Yaskawa INFORM job: KRIS3(-160_-90)54.JBI

/JOB
//NAME KRIS3(-160_-90)54
//POS
///NPOS 266,266,266,20,0,0
///TOOL 0
///POSTYPE PULSE
///PULSE
C00000=-36470,-76528,-106815,19279,71473,77234
C00001=-136908,-99459,-124829,20670,71348,76391
C00002=-134470,-76528,-106815,19279,71473,77234
C00003=-159578,-94739,-111578,14965,102577,71346
C00004=-157566,-87256,-71357,3912,80960,68626
C00005=-176880,-68125,-57902,5422,83635,62119
C00006=-177907,-68461,-55745,5507,82211,61705
C00007=-177907,-68063,-54493,5513,81648,61681
C00008=-177907,-68139,-54730,5512,81754,61686
C00009=-178677,-69433,-55362,5571,81531,61412
C00010=-178017,-68613,-55721,5516,82126,61665
C00011=-169648,-85474,-89038,4887,93378,64966
C00012=-163611,-44630,-68122,4506,101126,67267
C00013=-165231,-48362,-64740,4579,97228,66587
C00014=-165334,-48746,-64513,4584,96897,66540
C00015=-165334,-48893,-63576,4578,96247,66515
C00016=-165334,-48863,-63784,4579,96390,66520
C00017=-165646,-49802,-64330,4606,96263,66409
C00018=-165334,-48746,-64513,4584,96897,66540
C00019=-140979,-108094,-110643,2385,93763,74547
C00020=-140979,-108094,-110643,2385,93763,74547
C00021=-140979,-108094,-110643,2385,93763,74547
C00022=-140979,-108094,-110643,2385,93763,74547
C00023=-140979,-108246,-109289,2383,92853,74530
C00024=-140979,-108231,-109453,2383,92961,74533
C00025=-141280,-110659,-110301,2409,92244,74420
C00026=-140979,-108094,-110643,2385,93763,74547
C00027=-156700,-55897,-85418,-8720,99373,67438
C00028=-156898,-58036,-83987,-8629,97394,67513
C00029=-156898,-58722,-82817,-8603,96332,67586
C00030=-156898,-58622,-82997,-8608,96491,67574
C00031=-157341,-60416,-83948,-8523,96115,67457
C00032=-156898,-58036,-83987,-8629,97394,67513
C00033=-161369,-86849,-99090,4273,98390,67906
C00034=-167909,-84037,-82934,-3708,84523,64877
C00035=-168571,-85124,-82512,-3609,83677,64677
C00036=-168571,-84898,-80901,-3613,82804,64704
C00037=-168571,-84936,-81149,-3613,82937,64700
C00038=-169203,-86467,-81802,-3516,82525,64499
C00039=-168571,-85124,-82512,-3609,83677,64677
C00040=-165600,-121955,-98284,-4061,74695,65975
C00041=-174461,-109455,-70225,-9835,59183,64105
C00042=-175080,-109402,-69148,-9749,58483,63930
C00043=-175080,-108469,-67668,-9792,58058,63969
C00044=-175080,-108628,-67921,-9785,58130,63962
C00045=-176152,-109889,-68298,-9565,57596,63593
C00046=-175080,-109402,-69148,-9749,58483,63930
C00047=-145436,-132582,-96247,-390,75065,72870
C00048=-145436,-132678,-96385,-390,75101,72870
C00049=-145436,-153478,-122593,-390,33069,72870
C00050=-145436,-153478,-122593,-390,33069,72870
C00051=-145875,-137224,-99164,-151,44123,76557
C00052=-145875,-137224,-99164,3186,26783,75636
C00053=-145875,-137224,-99164,3186,26783,75636
C00054=-126920,-141995,-100488,-14842,27437,88451
C00055=-126921,-139435,-97257,-15195,26791,88624
C00056=-126921,-140260,-98306,-15082,27005,88567
C00057=-126657,-136107,-97292,-14665,28515,88375
C00058=-126920,-141995,-100488,-14842,27437,88451
C00059=-153689,-122615,-92358,-7246,28662,82796
C00060=-153689,-122359,-91923,-7277,28527,82812
C00061=-153689,-121251,-90046,-7417,27945,82882
C00062=-153689,-121596,-90629,-7373,28125,82859
C00063=-152562,-118169,-89603,-8504,29355,83484
C00064=-153689,-122359,-91923,-7277,28527,82812
C00065=-153734,-144670,-102026,12528,26386,79802
C00066=-148920,-141423,-91163,14854,15551,80235
C00067=-148967,-137496,-86916,15534,14983,79917
C00068=-147891,-134819,-86332,12174,15793,81580
C00069=-148428,-136185,-86633,13817,15374,80764
C00070=-148428,-134667,-84751,14154,15007,80609
C00071=-149705,-139389,-87494,17948,14535,78726
C00072=-140769,-160579,-91179,72763,19950,46602
C00073=-129302,-154781,-89703,59410,13959,54584
C00074=-128993,-152913,-89439,56337,14227,56040
C00075=-129214,-154274,-89633,58559,14027,54988
C00076=-129214,-151990,-87339,59384,13900,54610
C00077=-129539,-156129,-91089,59119,14177,54682
C00078=-130002,-156587,-91482,58522,14566,54861
C00079=-131612,-152018,-92345,56188,18115,55777
C00080=-137260,-138866,-133764,10166,31487,76482
C00081=-31464,-162597,-133764,10166,12061,76482
C00082=11401,-148032,-125425,11667,35640,75771
C00083=126225,-114648,-117375,36487,17100,65054
C00084=160935,-140983,-109640,13468,75088,74332
C00085=169853,-118963,-84593,12681,69660,-86771
C00086=166041,-110678,-74459,13320,68331,-88303
C00087=166223,-108797,-70951,13405,67140,-88373
C00088=166223,-107663,-69097,13458,66595,-88438
C00089=166223,-107867,-69431,13449,66693,-88427
C00090=167322,-109580,-69957,13369,65975,-88109
C00091=166243,-109210,-71582,13386,67309,-88347
C00092=169217,-106350,-70409,12947,67561,-87233
C00093=169217,-106256,-70250,12951,67512,-87238
C00094=169217,-105112,-68312,13006,66921,-87306
C00095=169217,-105283,-68599,12998,67008,-87297
C00096=170397,-106999,-69102,12897,66265,-86949
C00097=167930,-107758,-71144,13135,67501,-87709
C00098=168330,-125239,-100831,12460,76505,-86600
C00099=155830,-85289,-85709,13656,89459,-89593
C00100=155617,-85922,-82565,13677,87294,-89905
C00101=155617,-85683,-81004,13681,86480,-89993
C00102=155617,-85728,-81276,13680,86620,-89979
C00103=156391,-88450,-82422,13606,85816,-89798
C00104=155763,-86416,-82528,13661,87001,-89886
C00105=155923,-87175,-84120,13644,87549,-89771
C00106=155609,-85916,-82709,13676,87386,-89897
C00107=155609,-85729,-81437,13679,86718,-89971
C00108=155609,-85763,-81652,13678,86829,-89960
C00109=156185,-87803,-82513,13623,86229,-89826
C00110=155614,-85958,-82864,13674,87458,-89888
C00111=155923,-85281,-100905,13881,98543,-88548
C00112=155518,-83496,-100141,13947,99043,-88626
C00113=155616,-85272,-96985,13818,96251,-88909
C00114=155616,-85497,-96194,13797,95664,-88975
C00115=155616,-85451,-96366,13801,95791,-88960
C00116=156253,-88112,-97488,13709,95029,-88829
C00117=155726,-85538,-97830,13817,96606,-88830
C00118=154682,-87233,-101845,-693,104782,-88208
C00119=154465,-87160,-99128,-683,103145,-88271
C00120=154465,-87414,-98317,-682,102513,-88268
C00121=154465,-87352,-98526,-682,102673,-88268
C00122=154959,-89527,-99446,-690,102126,-88098
C00123=154682,-87831,-100410,-689,103591,-88201
C00124=156826,-87943,-103938,-737,105722,-87490
C00125=169505,-149944,-134809,-912,70958,-83129
C00126=169505,-149944,-134809,-912,70958,-83129
C00127=146455,-149944,-134809,-912,70958,-83129
C00128=112795,-148984,-134809,-2190,51374,-83129
C00129=111873,-164583,-130328,-1851,32186,-83318
C00130=111990,-161657,-129363,-1933,33097,-83272
C00131=111990,-159262,-126784,-1952,32742,-83264
C00132=111990,-160059,-127654,-1945,32868,-83268
C00133=112299,-153448,-126010,-2148,35260,-83152
C00134=111990,-161657,-129363,-1933,33097,-83272
C00135=102316,-143967,-116427,-74,34870,-80922
C00136=99836,-142438,-115626,2468,35200,-82353
C00137=99836,-141233,-113779,2484,34686,-82371
C00138=99836,-141783,-114624,2469,34923,-82363
C00139=100593,-136543,-113201,1615,36721,-81883
C00140=99836,-142438,-115626,2468,35200,-82353
C00141=118387,-195834,-126913,-32547,17814,-63683
C00142=108593,-194497,-126695,-13927,15739,-73675
C00143=111966,-142030,-104659,-11098,25227,-74939
C00144=111966,-142030,-104659,-11098,25227,-74939
C00145=112273,-138108,-103670,-10972,26650,-74986
C00146=112073,-140034,-103439,-11138,25510,-74915
C00147=112073,-138675,-101608,-11314,25090,-74828
C00148=112073,-140034,-103439,-11138,25510,-74915
C00149=133655,-153199,-106556,-41260,27910,-58399
C00150=149006,-93113,-100988,-5479,101691,-74295
C00151=149599,-96300,-103483,-5484,101628,-74092
C00152=92708,-143079,-100433,-810,17215,-88150
C00153=104933,-161562,-117451,-25070,27012,-78745
C00154=144107,-163968,-117280,-59568,38890,-55519
C00155=142578,-151510,-110599,-56645,39227,-57342
C00156=163022,-96736,-99152,22139,103253,-76925
C00157=162158,-93804,-96763,22109,103515,-77196
C00158=91813,-144765,-105961,-12434,16680,-86696
C00159=114692,-179984,-119020,-69502,19928,-58132
C00160=114692,-179984,-119020,-69502,19928,-58132
C00161=114692,-179984,-119020,-69502,19928,-58132
C00162=114692,-192492,-127590,-72579,19523,-56674
C00163=114692,-192492,-127590,-72579,19523,-56674
C00164=118502,-172484,-110233,-52609,25212,-65150
C00165=171509,-133648,-100111,-8061,78079,-67623
C00166=179980,-112353,-73580,-8533,73608,-64392
C00167=173099,-95941,-66024,-2428,83140,-67643
C00168=163006,-94576,-83573,21494,95359,-78388
C00169=162142,-91714,-81191,21448,95589,-78662
C00170=161519,-105438,-69378,-2986,79942,-71470
C00171=161519,-107811,-73451,-2977,81228,-71500
C00172=162580,-105162,-72246,8409,75537,-72147
C00173=166978,-101333,-67887,8237,74379,-70700
C00174=163006,-94576,-83573,21494,95359,-78388
C00175=162142,-91714,-81191,21448,95589,-78662
C00176=176806,-91826,-64313,7611,76084,-67180
C00177=169252,-115124,-101169,7872,87423,-69075
C00178=154261,-79873,-81468,8571,94879,-73696
C00179=156149,-79526,-78849,8481,93264,-73164
C00180=163006,-94576,-83573,21494,95359,-78388
C00181=162142,-91714,-81191,21448,95589,-78662
C00182=164231,-71322,-75012,8167,94272,-70347
C00183=163718,-69809,-76291,8220,95872,-70416
C00184=152145,-81088,-82167,2065,97703,-74759
C00185=153873,-81294,-80148,2070,96313,-74194
C00186=163006,-94576,-83573,21494,95359,-78388
C00187=162142,-91714,-81191,21448,95589,-78662
C00188=144574,-87616,-82877,1978,94978,-77376
C00189=144574,-84995,-103251,2104,108854,-77145
C00190=151765,-102418,-106955,-5657,95758,-75438
C00191=152438,-102405,-104678,-5690,94416,-75154
C00192=163006,-94576,-83573,21494,95359,-78388
C00193=162142,-91714,-81191,21448,95589,-78662
C00194=141196,-110717,-107651,-4757,91265,-78794
C00195=143989,-108966,-109417,-5008,93413,-77941
C00196=143223,-109509,-108756,8615,88663,-77081
C00197=144525,-109134,-106137,8437,87124,-76746
C00198=163006,-94576,-83573,21494,95359,-78388
C00199=162142,-91714,-81191,21448,95589,-78662
C00200=155521,-99997,-102811,6821,88724,-72955
C00201=144143,-146387,-128453,8544,81812,-77235
C00202=130399,-165491,-128261,-582,73715,-81342
C00203=149731,-158641,-113843,14975,70738,69794
C00204=149731,-158641,-113843,14975,70738,69794
C00205=126225,-114648,-117375,36487,17100,65054
C00206=118781,-153853,-134406,32592,23357,65054
C00207=12470,-167083,-125425,11667,16324,75771
C00208=-137258,-84249,-120477,10166,64820,76482
C00209=-160540,-100857,-113063,23155,68829,67581
C00210=-182830,-114405,-112845,16003,91175,61677
C00211=-183790,-123536,-112279,16086,86512,60735
C00212=-173371,-96838,-101602,8067,99830,65021
C00213=-158743,-95268,-103371,5812,102972,69826
C00214=-157888,-92366,-100981,5813,102933,70115
C00215=-163928,-110855,-106734,7756,94909,67922
C00216=-164197,-113877,-111682,7800,96401,67923
C00217=-173870,-143306,-120553,7913,87764,64082
C00218=-171816,-118751,-98057,3590,91441,64891
C00219=-175172,-115602,-92589,3406,89844,63709
C00220=-158755,-94787,-86481,-976,103949,69303
C00221=-157900,-91912,-84097,-841,103969,69603
C00222=-163756,-128157,-96341,3996,85186,67438
C00223=-163756,-130674,-100363,3993,86365,67475
C00224=-177254,-154866,-106204,3341,78153,62695
C00225=-194740,-128784,-79093,2289,75465,56815
C00226=-198284,-123329,-74228,2053,75365,55640
C00227=-158782,-86330,-62292,2348,97119,70521
C00228=-157926,-83586,-59872,2521,97014,70811
C00229=-186334,-135847,-76880,2902,70224,59482
C00230=-186334,-138981,-80518,2891,70851,59497
C00231=-202790,-114657,-73561,-7469,64730,55511
C00232=-205482,-109926,-69448,-7082,64394,54553
C00233=-158743,-95268,-103371,5812,102972,69826
C00234=-157888,-92366,-100981,5813,102933,70115
C00235=-208812,-100961,-65482,-8613,62862,53643
C00236=-188075,-151957,-103997,-12598,63075,61358
C00237=-175676,-115929,-94468,-13375,77380,64283
C00238=-178876,-108879,-88776,-12955,76978,63190
C00239=-158755,-94787,-86481,-976,103949,69303
C00240=-157900,-91912,-84097,-841,103969,69603
C00241=-187253,-94310,-83232,-11601,79689,59970
C00242=-178297,-108275,-107099,-12771,88378,62209
C00243=-165278,-79866,-95804,-14582,97947,65562
C00244=-166994,-82226,-93327,-14277,95001,65330
C00245=-158782,-86330,-62292,2348,97119,70521
C00246=-157926,-83586,-59872,2521,97014,70811
C00247=-172105,-74751,-88994,-16012,93362,63480
C00248=-166883,-83368,-97274,-16810,95013,65031
C00249=-148381,-154133,-120540,-18986,77988,74048
C00250=-148381,-154133,-120540,-18986,29025,74048
C00251=-148381,-154133,-120540,-18986,29025,74048
C00252=-148381,-154133,-120540,-18986,29025,74048
C00253=-148381,-154133,-120540,-635,27393,68347
C00254=-131809,-160671,-109428,-31686,20564,84507
C00255=-131822,-150264,-103689,-29313,22136,83370
C00256=-180653,-114218,-94091,32947,38431,50047
C00257=-160079,-162229,-113551,20584,20355,57319
C00258=-127848,-170739,-113822,25929,20694,59837
C00259=-98584,-145628,-105124,-27441,32859,85558
C00260=-101312,-135763,-98504,-24330,32920,83709
C00261=-155537,-127424,-96398,29935,38582,51900
C00262=-162526,-150393,-107796,38053,37342,46820
C00263=-161637,-148332,-107324,36893,37578,47548
C00264=-136473,-81821,-106853,20577,68974,75046
C00265=-36470,-76528,-106815,19279,71473,77234
BC00000=295325,674563,1075175
BC00001=353535,857279,1075175
BC00002=353535,895977,1075175
BC00003=353535,975867,1075175
BC00004=382950,976989,1075175
BC00005=382950,976989,1075175
BC00006=382950,976989,1075175
BC00007=382950,976989,1075175
BC00008=382950,976989,1075175
BC00009=382950,976989,1075175
BC00010=382950,976989,1075175
BC00011=382950,976989,1075172
BC00012=382950,976989,1075172
BC00013=382950,976989,1075172
BC00014=382950,976989,1075172
BC00015=382950,976989,1075172
BC00016=382950,976989,1075172
BC00017=382950,976989,1075172
BC00018=382950,976989,1075172
BC00019=329549,1006497,1075175
BC00020=329549,1029947,1075175
BC00021=325179,1029723,1057241
BC00022=324419,1030107,1053762
BC00023=324419,1030107,1053762
BC00024=324419,1030107,1053762
BC00025=324419,1030107,1053762
BC00026=324419,1030107,1053762
BC00027=326367,1006363,1075175
BC00028=326367,1006363,1075175
BC00029=326367,1006363,1075175
BC00030=326367,1006363,1075175
BC00031=326367,1006363,1075175
BC00032=326367,1006363,1075175
BC00033=324712,1006363,1075175
BC00034=324712,1006363,1075175
BC00035=324712,1006363,1075175
BC00036=324712,1006363,1075175
BC00037=324712,1006363,1075175
BC00038=324712,1006363,1075175
BC00039=324712,1006363,1075175
BC00040=324712,1006363,1075175
BC00041=324712,1006363,1075175
BC00042=324712,1006363,1075175
BC00043=324712,1006363,1075175
BC00044=324712,1006363,1075175
BC00045=324712,1006363,1075175
BC00046=324712,1006363,1075175
BC00047=334035,1006363,1075175
BC00048=334035,1006363,1075175
BC00049=334035,960963,1075175
BC00050=369533,796939,1075175
BC00051=369533,796939,1075175
BC00052=324907,880615,715339
BC00053=299333,903943,711615
BC00054=299333,903943,711615
BC00055=299333,903943,711613
BC00056=299333,903943,711613
BC00057=299333,903943,711613
BC00058=299333,903943,711615
BC00059=299333,903943,711615
BC00060=299333,903943,711615
BC00061=299333,903943,711615
BC00062=299333,903943,711615
BC00063=299333,903943,711615
BC00064=299333,903943,711615
BC00065=327028,893674,717250
BC00066=327028,893674,706960
BC00067=327028,893674,706958
BC00068=327028,893674,706958
BC00069=327028,893674,706958
BC00070=327028,893674,706958
BC00071=327028,893674,706958
BC00072=321055,903094,706958
BC00073=321055,903094,706958
BC00074=321055,903094,706958
BC00075=321055,903094,706958
BC00076=321055,903094,706958
BC00077=321055,903094,706958
BC00078=307667,855149,971272
BC00079=312219,773310,1067430
BC00080=353816,923989,1075175
BC00081=379773,1126391,1075175
BC00082=398190,1030285,1075175
BC00083=312632,1138057,1075175
BC00084=340753,1115300,1075175
BC00085=340766,1114848,1075175
BC00086=340766,1114848,1075175
BC00087=340766,1114848,1075175
BC00088=340766,1114848,1075175
BC00089=340766,1114848,1075175
BC00090=340766,1114848,1075175
BC00091=340766,1114848,1075175
BC00092=373830,1114848,1075175
BC00093=373830,1114848,1075175
BC00094=373830,1114848,1075175
BC00095=373830,1114848,1075175
BC00096=373830,1114848,1075175
BC00097=373830,1114848,1075175
BC00098=373830,1114848,1075175
BC00099=373830,1114848,1075175
BC00100=373830,1114848,1075175
BC00101=373830,1114848,1075175
BC00102=373830,1114848,1075175
BC00103=373830,1114848,1075175
BC00104=373830,1114848,1075175
BC00105=340054,1114848,1075175
BC00106=340054,1115648,1071892
BC00107=340054,1115648,1071892
BC00108=340054,1115648,1071892
BC00109=340054,1115648,1071892
BC00110=340054,1115648,1071892
BC00111=340054,1115648,1073754
BC00112=340054,1089258,1073754
BC00113=340054,1089258,1073754
BC00114=340054,1089258,1073754
BC00115=340054,1089258,1073754
BC00116=340054,1089258,1073754
BC00117=340054,1089258,1073754
BC00118=340054,1089258,1073754
BC00119=340054,1089258,1073754
BC00120=340054,1089258,1073754
BC00121=340054,1089258,1073754
BC00122=340054,1089258,1073754
BC00123=340054,1089258,1073754
BC00124=340054,1089258,1073754
BC00125=340054,1089258,1073754
BC00126=387158,1273206,1073754
BC00127=354276,1245348,772198
BC00128=302489,1244324,601573
BC00129=305225,1224612,556934
BC00130=305225,1224612,556934
BC00131=305225,1224612,556934
BC00132=305225,1224612,556934
BC00133=305225,1224612,556934
BC00134=305225,1224612,556934
BC00135=332360,1224612,614061
BC00136=332360,1224612,614061
BC00137=332360,1224612,614060
BC00138=332360,1224612,614060
BC00139=332360,1224612,614060
BC00140=332360,1224612,614061
BC00141=332360,1224612,614061
BC00142=276926,1224612,614061
BC00143=288820,1246847,685550
BC00144=272480,1241151,623068
BC00145=272480,1241151,623068
BC00146=272480,1241151,623068
BC00147=272480,1241151,623068
BC00148=272480,1241151,623068
BC00149=264384,1231863,612337
BC00150=348912,1090234,1075175
BC00151=348912,1090234,1075175
BC00152=264384,1231863,612337
BC00153=270263,1230158,610880
BC00154=307096,1219473,601753
BC00155=307096,1219473,601753
BC00156=322536,1051450,1075175
BC00157=322536,1051450,1075175
BC00158=307096,1219473,601753
BC00159=307096,1219473,601753
BC00160=307096,1219473,601753
BC00161=285358,1283082,784261
BC00162=285358,1283082,1042648
BC00163=308804,1178054,1042648
BC00164=314237,1167311,1048176
BC00165=340766,1114849,1075169
BC00166=340766,1114849,1075169
BC00167=340766,1114849,1075169
BC00168=322462,1078251,1075175
BC00169=322462,1078251,1075175
BC00170=340766,1114849,1075169
BC00171=340766,1114849,1075169
BC00172=340766,1114849,1075169
BC00173=340766,1114849,1075169
BC00174=322462,1078251,1075175
BC00175=322462,1078251,1075175
BC00176=340766,1114849,1075169
BC00177=340766,1114849,1075169
BC00178=340766,1114849,1075169
BC00179=340766,1114849,1075169
BC00180=322462,1078251,1075175
BC00181=322462,1078251,1075175
BC00182=340766,1114849,1075169
BC00183=340766,1114849,1075169
BC00184=340766,1114849,1075169
BC00185=340766,1114849,1075169
BC00186=322462,1078251,1075175
BC00187=322462,1078251,1075175
BC00188=340766,1114849,1075169
BC00189=340766,1114849,1075169
BC00190=323476,1092417,1070465
BC00191=323476,1092417,1070465
BC00192=322462,1078251,1075175
BC00193=322462,1078251,1075175
BC00194=323476,1092417,1070465
BC00195=323476,1092417,1070465
BC00196=323476,1092417,1070465
BC00197=323476,1092417,1070465
BC00198=322462,1078251,1075175
BC00199=322462,1078251,1075175
BC00200=323476,1092417,1070465
BC00201=323476,1092417,1070465
BC00202=333441,1105345,1073176
BC00203=340753,1115300,1075175
BC00204=340753,1115300,1075175
BC00205=312632,1138057,1075175
BC00206=312632,1138057,1075175
BC00207=398190,1030285,1075175
BC00208=353817,923990,1075175
BC00209=381896,966588,1075175
BC00210=347402,1044565,1075172
BC00211=347402,1044565,1075172
BC00212=347402,1044565,1075172
BC00213=364655,1041006,1075175
BC00214=364655,1041006,1075175
BC00215=347402,1044565,1075172
BC00216=347622,1044563,1075172
BC00217=347622,1044563,1075172
BC00218=338568,1044451,1075174
BC00219=338569,1044452,1075171
BC00220=364774,1039056,1075175
BC00221=364774,1039056,1075175
BC00222=338569,1044452,1075171
BC00223=338569,1044452,1075171
BC00224=338569,1044452,1075171
BC00225=338569,1044452,1075171
BC00226=338569,1044452,1075171
BC00227=355520,1012445,1075175
BC00228=355520,1012445,1075175
BC00229=338569,1044452,1075171
BC00230=338569,1044452,1075171
BC00231=338569,1044452,1075171
BC00232=338569,1044452,1075171
BC00233=364655,1041006,1075175
BC00234=364655,1041006,1075175
BC00235=338569,1044452,1075171
BC00236=338569,1044452,1075171
BC00237=338569,1044452,1075171
BC00238=338569,1044452,1075171
BC00239=364774,1039056,1075175
BC00240=364774,1039056,1075175
BC00241=338569,1044452,1075171
BC00242=338569,1044452,1075171
BC00243=338569,1044452,1075171
BC00244=338569,1044452,1075171
BC00245=355520,1012445,1075175
BC00246=355520,1012445,1075175
BC00247=338569,1044452,1075171
BC00248=338569,1044452,1075171
BC00249=338569,1044452,1075171
BC00250=378565,961750,1075171
BC00251=386061,798644,1075171
BC00252=386061,798644,789316
BC00253=347571,884540,659815
BC00254=318020,909055,659815
BC00255=318020,909055,659815
BC00256=318020,909055,659815
BC00257=318020,909055,659815
BC00258=331358,890408,659815
BC00259=316626,888097,659815
BC00260=316626,888097,659815
BC00261=316626,888097,659815
BC00262=316626,888097,659815
BC00263=316626,758293,915546
BC00264=350814,688495,1063408
BC00265=295325,674563,1075175
EC00000=-1418945,-556475
EC00001=-1418945,-556475
EC00002=-1418945,-556475
EC00003=-1418945,-556475
EC00004=-1418945,-556475
EC00005=-1418945,-556475
EC00006=-1418945,-556475
EC00007=-1418945,-556475
EC00008=-1418945,-556475
EC00009=-1418945,-556475
EC00010=-1418945,-556475
EC00011=-1418944,-556475
EC00012=-1418944,-556475
EC00013=-1418944,-556475
EC00014=-1418944,-556475
EC00015=-1418944,-556475
EC00016=-1418944,-556475
EC00017=-1418944,-556475
EC00018=-1418944,-556475
EC00019=-1418945,-556475
EC00020=-1418945,-556475
EC00021=-1418945,-556475
EC00022=-1418945,-556475
EC00023=-1418945,-556475
EC00024=-1418945,-556475
EC00025=-1418945,-556475
EC00026=-1418945,-556475
EC00027=-1418945,-556475
EC00028=-1418945,-556475
EC00029=-1418945,-556475
EC00030=-1418945,-556475
EC00031=-1418945,-556475
EC00032=-1418945,-556475
EC00033=-1418945,-556475
EC00034=-1418945,-556475
EC00035=-1418945,-556475
EC00036=-1418945,-556475
EC00037=-1418945,-556475
EC00038=-1418945,-556475
EC00039=-1418945,-556475
EC00040=-1418945,-556475
EC00041=-1418945,-556475
EC00042=-1418945,-556475
EC00043=-1418945,-556475
EC00044=-1418945,-556475
EC00045=-1418945,-556475
EC00046=-1418945,-556475
EC00047=-1418945,-556475
EC00048=-1418945,-556475
EC00049=-1418945,-556475
EC00050=-1418945,-556475
EC00051=-1418945,-556475
EC00052=-1418945,-556475
EC00053=-1418945,-556475
EC00054=-1418945,-556475
EC00055=-1418944,-556475
EC00056=-1418944,-556475
EC00057=-1418944,-556475
EC00058=-1418945,-556475
EC00059=-1418945,-556475
EC00060=-1418945,-556475
EC00061=-1418945,-556475
EC00062=-1418945,-556475
EC00063=-1418945,-556475
EC00064=-1418945,-556475
EC00065=-1418945,-556475
EC00066=-1418945,-556475
EC00067=-1418945,-556475
EC00068=-1418945,-556475
EC00069=-1418945,-556475
EC00070=-1418945,-556475
EC00071=-1418945,-556475
EC00072=-1418945,-556475
EC00073=-1418945,-556475
EC00074=-1418945,-556475
EC00075=-1418945,-556475
EC00076=-1418945,-556475
EC00077=-1418945,-556475
EC00078=-1418945,-556475
EC00079=-1418945,-556475
EC00080=-1418945,-556475
EC00081=-1418945,-556475
EC00082=-1595090,-3837
EC00083=-1773681,556475
EC00084=-1773681,556475
EC00085=-1773681,556475
EC00086=-1773681,556475
EC00087=-1773681,556475
EC00088=-1773681,556475
EC00089=-1773681,556475
EC00090=-1773681,556475
EC00091=-1773681,556475
EC00092=-1773681,556475
EC00093=-1773681,556475
EC00094=-1773681,556475
EC00095=-1773681,556475
EC00096=-1773681,556475
EC00097=-1773681,556475
EC00098=-1773681,556475
EC00099=-1773681,556475
EC00100=-1773681,556475
EC00101=-1773681,556475
EC00102=-1773681,556475
EC00103=-1773681,556475
EC00104=-1773681,556475
EC00105=-1773681,556475
EC00106=-1773681,556475
EC00107=-1773681,556475
EC00108=-1773681,556475
EC00109=-1773681,556475
EC00110=-1773681,556475
EC00111=-1773681,556475
EC00112=-1773681,556475
EC00113=-1773681,556475
EC00114=-1773681,556475
EC00115=-1773681,556475
EC00116=-1773681,556475
EC00117=-1773681,556475
EC00118=-1773681,556475
EC00119=-1773681,556475
EC00120=-1773681,556475
EC00121=-1773681,556475
EC00122=-1773681,556475
EC00123=-1773681,556475
EC00124=-1773681,556475
EC00125=-1773681,556475
EC00126=-1773681,556475
EC00127=-1773681,556475
EC00128=-1773681,556475
EC00129=-1773681,556475
EC00130=-1773681,556475
EC00131=-1773681,556475
EC00132=-1773681,556475
EC00133=-1773681,556475
EC00134=-1773681,556475
EC00135=-1773681,556475
EC00136=-1773681,556475
EC00137=-1773682,556474
EC00138=-1773682,556474
EC00139=-1773682,556474
EC00140=-1773681,556475
EC00141=-1773681,556475
EC00142=-1773681,556475
EC00143=-1773681,556475
EC00144=-1773681,556475
EC00145=-1773681,556475
EC00146=-1773681,556475
EC00147=-1773681,556475
EC00148=-1773681,556475
EC00149=-1773681,556475
EC00150=-1773681,556475
EC00151=-1773681,556475
EC00152=-1773681,556475
EC00153=-1773681,556475
EC00154=-1773681,556475
EC00155=-1773681,556475
EC00156=-1773681,556475
EC00157=-1773681,556475
EC00158=-1773681,556475
EC00159=-1773681,556475
EC00160=-1773681,556475
EC00161=-1773681,556475
EC00162=-1773681,556475
EC00163=-1773681,556475
EC00164=-1773681,556475
EC00165=-1773683,556473
EC00166=-1773683,556473
EC00167=-1773683,556473
EC00168=-1773681,556475
EC00169=-1773681,556475
EC00170=-1773683,556473
EC00171=-1773683,556473
EC00172=-1773683,556473
EC00173=-1773683,556473
EC00174=-1773681,556475
EC00175=-1773681,556475
EC00176=-1773683,556473
EC00177=-1773683,556473
EC00178=-1773683,556473
EC00179=-1773683,556473
EC00180=-1773681,556475
EC00181=-1773681,556475
EC00182=-1773683,556473
EC00183=-1773683,556473
EC00184=-1773683,556473
EC00185=-1773683,556473
EC00186=-1773681,556475
EC00187=-1773681,556475
EC00188=-1773683,556473
EC00189=-1773683,556473
EC00190=-1773683,556473
EC00191=-1773683,556473
EC00192=-1773681,556475
EC00193=-1773681,556475
EC00194=-1773683,556473
EC00195=-1773683,556473
EC00196=-1773683,556473
EC00197=-1773683,556473
EC00198=-1773681,556475
EC00199=-1773681,556475
EC00200=-1773683,556473
EC00201=-1773683,556473
EC00202=-1773683,556473
EC00203=-1773681,556475
EC00204=-1773681,556475
EC00205=-1773681,556475
EC00206=-1773681,556475
EC00207=-1595090,-3837
EC00208=-1418947,-556468
EC00209=-1418945,-556475
EC00210=-1418944,-556475
EC00211=-1418944,-556475
EC00212=-1418944,-556475
EC00213=-1418945,-556475
EC00214=-1418945,-556475
EC00215=-1418944,-556475
EC00216=-1418944,-556475
EC00217=-1418944,-556475
EC00218=-1418945,-556475
EC00219=-1418944,-556475
EC00220=-1418945,-556475
EC00221=-1418945,-556475
EC00222=-1418944,-556475
EC00223=-1418944,-556475
EC00224=-1418944,-556475
EC00225=-1418944,-556475
EC00226=-1418944,-556475
EC00227=-1418945,-556475
EC00228=-1418945,-556475
EC00229=-1418944,-556475
EC00230=-1418944,-556475
EC00231=-1418944,-556475
EC00232=-1418944,-556475
EC00233=-1418945,-556475
EC00234=-1418945,-556475
EC00235=-1418944,-556475
EC00236=-1418944,-556475
EC00237=-1418944,-556475
EC00238=-1418944,-556475
EC00239=-1418945,-556475
EC00240=-1418945,-556475
EC00241=-1418944,-556475
EC00242=-1418944,-556475
EC00243=-1418944,-556475
EC00244=-1418944,-556475
EC00245=-1418945,-556475
EC00246=-1418945,-556475
EC00247=-1418944,-556475
EC00248=-1418944,-556475
EC00249=-1418944,-556475
EC00250=-1418944,-556475
EC00251=-1418944,-556475
EC00252=-1418944,-556475
EC00253=-1418944,-556475
EC00254=-1418944,-556475
EC00255=-1418944,-556475
EC00256=-1418944,-556475
EC00257=-1418944,-556475
EC00258=-1418944,-556475
EC00259=-1418944,-556475
EC00260=-1418944,-556475
EC00261=-1418944,-556475
EC00262=-1418944,-556475
EC00263=-1418944,-556475
EC00264=-1418945,-556475
EC00265=-1418945,-556475
///POSTYPE BASE
///RECTAN
///RCONF 0,0,0,0,0,0,0,0,0,0,0,0,0,0,0,0,0,0,0,0,0,0,0,0
P00006=0.232,-0.094,-1.480,0.0000,0.0000,0.0000
P00021=-0.225,-6.128,-0.405,0.0000,0.0000,0.0000
P00022=0.232,-0.094,-1.480,0.0000,0.0000,0.0000
P00023=0.143,-0.036,0.682,0.0000,0.0000,0.0000
P00024=0.145,-0.552,1.326,0.0000,0.0000,0.0000
P00025=-2.003,0.006,0.728,0.0000,0.0000,0.0000
P00026=0.562,-0.002,-0.337,0.0000,0.0000,0.0000
P00027=-0.746,0.015,-9.096,0.0000,0.0000,0.0000
P00028=-2.237,-0.018,-7.702,0.0000,0.0000,0.0000
P00029=-2.156,-0.086,-4.681,0.0000,0.0000,0.0000
P00030=5.926,-4.294,-1.390,0.0000,0.0000,0.0000
P00031=1.853,-0.001,-1.549,0.0000,0.0000,0.0000
P00032=1.957,0.503,-7.217,0.0000,0.0000,0.0000
///RCONF 0,0,0,0,1,0,0,0,0,0,0,0,0,0,0,0,0,0,0,0,0,0,0,0
P00033=-0.123,0.612,-5.012,0.0000,0.0000,0.0000
///RCONF 0,0,0,0,0,0,0,0,0,0,0,0,0,0,0,0,0,0,0,0,0,0,0,0
P00034=-0.304,0.773,-2.693,0.0000,0.0000,0.0000
P00035=2.817,0.591,-1.622,0.0000,0.0000,0.0000
P00036=-1.108,-0.829,1.850,0.0000,0.0000,0.0000
P00037=0.023,0.937,-2.677,0.0000,0.0000,0.0000
P00038=0.158,-1.133,-1.952,0.0000,0.0000,0.0000
P00039=0.012,-3.081,-0.106,0.0000,0.0000,0.0000
//INST
///DATE 2024/05/16 22:54
///ATTR SC,RW
///GROUP1 RB1,BS1
///GROUP2 ST1
NOP
MOVJ C00000 BC00000 VJ=100.00  +MOVJ EC00000 VJ=100.00
'MUZYLO 260124 START
MOVJ C00001 BC00001 VJ=100.00  +MOVJ EC00001 VJ=100.00
MOVJ C00002 BC00002 VJ=100.00  +MOVJ EC00002 VJ=100.00
MOVJ C00003 BC00003 VJ=100.00  +MOVJ EC00003 VJ=100.00
'Path S1422
SFTOF3D
MOVJ C00004 BC00004 VJ=100.00  +MOVJ EC00004 VJ=100.00
MOVL C00005 BC00005 V=400.0  +MOVJ EC00005 VJ=100.00
SMOVL C00006 BC00006 V=100.0  +MOVJ EC00006
SREFP 3 C00007 BC00007  +REFP EC00007
CALL JOB:SEARCH-R1-S13D
SET P021 P006
SFTON3D P021
SMOVL C00008 BC00008 V=100.0  +MOVJ EC00008
SREFP 3 C00009 BC00009  +REFP EC00009
CALL JOB:SEARCH-R1-S13D
SET P021 P006
SFTON3D P021
SMOVL C00010 BC00010 V=100.0  +MOVJ EC00010
MOVL C00011 BC00011 V=400.0  +MOVJ EC00011 VJ=100.00
MOVL C00012 BC00012 V=1000.0  +MOVJ EC00012 VJ=100.00
MOVJ C00013 BC00013 VJ=100.00  +MOVJ EC00013 VJ=100.00
'Path S1423
SFTOF3D
SMOVL C00014 BC00014 V=100.0  +MOVJ EC00014
SREFP 3 C00015 BC00015  +REFP EC00015
CALL JOB:SEARCH-R1-S13D
SET P022 P006
SFTON3D P022
SMOVL C00016 BC00016 V=100.0  +MOVJ EC00016
SREFP 3 C00017 BC00017  +REFP EC00017
CALL JOB:SEARCH-R1-S13D
SET P022 P006
SFTON3D P022
SMOVL C00018 BC00018 V=100.0  +MOVJ EC00018
MOVL C00019 BC00019 V=400.0  +MOVJ EC00019 VJ=100.00
MOVL C00020 BC00020 V=1000.0  +MOVJ EC00020 VJ=100.00
MOVJ C00021 BC00021 VJ=100.00  +MOVJ EC00021 VJ=100.00
'Path S1424
SFTOF3D
SMOVL C00022 BC00022 V=100.0  +MOVJ EC00022
SREFP 3 C00023 BC00023  +REFP EC00023
CALL JOB:SEARCH-R1-S13D
SET P023 P006
SFTON3D P023
SMOVL C00024 BC00024 V=100.0  +MOVJ EC00024
SREFP 3 C00025 BC00025  +REFP EC00025
CALL JOB:SEARCH-R1-S13D
SET P023 P006
SFTON3D P023
SMOVL C00026 BC00026 V=100.0  +MOVJ EC00026
MOVL C00027 BC00027 V=400.0  +MOVJ EC00027 VJ=100.00
SMOVL C00028 BC00028 V=100.0  +MOVJ EC00028
SREFP 3 C00029 BC00029  +REFP EC00029
CALL JOB:SEARCH-R1-S13D
SET P024 P006
SFTON3D P024
SMOVL C00030 BC00030 V=100.0  +MOVJ EC00030
SREFP 3 C00031 BC00031  +REFP EC00031
CALL JOB:SEARCH-R1-S13D
SET P024 P006
SFTON3D P024
SMOVL C00032 BC00032 V=100.0  +MOVJ EC00032
MOVL C00033 BC00033 V=400.0  +MOVJ EC00033 VJ=100.00
MOVL C00034 BC00034 V=1000.0  +MOVJ EC00034 VJ=100.00
'Path S1423
SFTOF3D
SMOVL C00035 BC00035 V=100.0  +MOVJ EC00035
SREFP 3 C00036 BC00036  +REFP EC00036
CALL JOB:SEARCH-R1-S13D
SET P025 P006
SFTON3D P025
SMOVL C00037 BC00037 V=100.0  +MOVJ EC00037
SREFP 3 C00038 BC00038  +REFP EC00038
CALL JOB:SEARCH-R1-S13D
SET P025 P006
SFTON3D P025
SMOVL C00039 BC00039 V=100.0  +MOVJ EC00039
MOVL C00040 BC00040 V=400.0  +MOVJ EC00040 VJ=100.00
MOVL C00041 BC00041 V=1000.0  +MOVJ EC00041 VJ=100.00
'Path S1424
SFTOF3D
SMOVL C00042 BC00042 V=100.0  +MOVJ EC00042
SREFP 3 C00043 BC00043  +REFP EC00043
CALL JOB:SEARCH-R1-S13D
SET P026 P006
SFTON3D P026
SMOVL C00044 BC00044 V=100.0  +MOVJ EC00044
SREFP 3 C00045 BC00045  +REFP EC00045
CALL JOB:SEARCH-R1-S13D
SET P026 P006
SFTON3D P026
SMOVL C00046 BC00046 V=100.0  +MOVJ EC00046
MOVL C00047 BC00047 V=400.0  +MOVJ EC00047 VJ=100.00
MOVJ C00048 BC00048 VJ=50.00  +MOVJ EC00048 VJ=50.00
MOVJ C00049 BC00049 VJ=100.00  +MOVJ EC00049 VJ=50.00
MOVJ C00050 BC00050 VJ=100.00  +MOVJ EC00050 VJ=50.00
MOVJ C00051 BC00051 VJ=100.00  +MOVJ EC00051 VJ=50.00
MOVJ C00052 BC00052 VJ=100.00  +MOVJ EC00052 VJ=50.00
MOVJ C00053 BC00053 VJ=100.00  +MOVJ EC00053 VJ=50.00
SFTOF3D
SMOVL C00054 BC00054 V=166.7  +MOVJ EC00054
SREFP 3 C00055 BC00055  +REFP EC00055
CALL JOB:SEARCH-R1-S13D
SET P027 P006
SFTON3D P027
SMOVL C00056 BC00056 V=100.0  +MOVJ EC00056
SREFP 3 C00057 BC00057  +REFP EC00057
CALL JOB:SEARCH-R1-S13D
SET P027 P006
SFTON3D P027
SMOVL C00058 BC00058 V=100.0  +MOVJ EC00058
SMOVL C00059 BC00059 V=416.7  +MOVJ EC00059
SFTOF3D
SMOVL C00060 BC00060 V=100.0  +MOVJ EC00060
SREFP 3 C00061 BC00061  +REFP EC00061
CALL JOB:SEARCH-R1-S13D
SET P028 P006
SFTON3D P028
SMOVL C00062 BC00062 V=100.0  +MOVJ EC00062
SREFP 3 C00063 BC00063  +REFP EC00063
CALL JOB:SEARCH-R1-S13D
SET P028 P006
SFTON3D P028
SMOVL C00064 BC00064 V=100.0  +MOVJ EC00064
SMOVL C00065 BC00065 V=416.7  +MOVJ EC00065
SMOVL C00066 BC00066 V=416.7  +MOVJ EC00066
SFTOF3D
SMOVL C00067 BC00067 V=100.0  +MOVJ EC00067
SREFP 3 C00068 BC00068  +REFP EC00068
CALL JOB:SEARCH-R1-S13D
SET P029 P006
SFTON3D P029
SMOVL C00069 BC00069 V=100.0  +MOVJ EC00069
SREFP 3 C00070 BC00070  +REFP EC00070
CALL JOB:SEARCH-R1-S13D
SET P029 P006
SFTON3D P029
SMOVL C00071 BC00071 V=100.0  +MOVJ EC00071
MOVJ C00072 BC00072 VJ=100.00  +MOVJ EC00072 VJ=50.00
SFTOF3D
SMOVL C00073 BC00073 V=83.3  +MOVJ EC00073
SREFP 3 C00074 BC00074  +REFP EC00074
CALL JOB:SEARCH-R1-S13D
SET P030 P006
SFTON3D P030
SMOVL C00075 BC00075 V=100.0  +MOVJ EC00075
SREFP 3 C00076 BC00076  +REFP EC00076
CALL JOB:SEARCH-R1-S13D
SET P030 P006
SFTON3D P030
SMOVL C00077 BC00077 V=100.0  +MOVJ EC00077
MOVL C00078 BC00078 V=1000.0  +MOVJ EC00078 VJ=100.00
'obrot
MOVJ C00079 BC00079 VJ=100.00  +MOVJ EC00079 VJ=100.00
MOVJ C00080 BC00080 VJ=100.00  +MOVJ EC00080 VJ=100.00
MOVJ C00081 BC00081 VJ=100.00  +MOVJ EC00081 VJ=100.00
MOVJ C00082 BC00082 VJ=100.00  +MOVJ EC00082 VJ=100.00
MOVJ C00083 BC00083 VJ=100.00  +MOVJ EC00083 VJ=100.00
MOVJ C00084 BC00084 VJ=100.00  +MOVJ EC00084 VJ=100.00
'Path S1077
SFTOF3D
MOVJ C00085 BC00085 VJ=100.00  +MOVJ EC00085 VJ=100.00
MOVL C00086 BC00086 V=400.0  +MOVJ EC00086 VJ=100.00
SMOVL C00087 BC00087 V=100.0  +MOVJ EC00087
SREFP 3 C00088 BC00088  +REFP EC00088
CALL JOB:SEARCH-R1-S13D
SET P031 P006
SFTON3D P031
SMOVL C00089 BC00089 V=100.0  +MOVJ EC00089
SREFP 3 C00090 BC00090  +REFP EC00090
CALL JOB:SEARCH-R1-S13D
SET P031 P006
SFTON3D P031
SMOVL C00091 BC00091 V=133.3  +MOVJ EC00091
SMOVL C00092 BC00092 V=666.7  +MOVJ EC00092 VJ=100.00
'Path S1078
SFTOF3D
SMOVL C00093 BC00093 V=100.0  +MOVJ EC00093
SREFP 3 C00094 BC00094  +REFP EC00094
CALL JOB:SEARCH-R1-S13D
SET P032 P006
SFTON3D P032
SMOVL C00095 BC00095 V=100.0  +MOVJ EC00095
SREFP 3 C00096 BC00096  +REFP EC00096
CALL JOB:SEARCH-R1-S13D
SET P032 P006
SFTON3D P032
SMOVL C00097 BC00097 V=100.0  +MOVJ EC00097
MOVL C00098 BC00098 V=1000.0  +MOVJ EC00098 VJ=100.00
'Path S1079
SFTOF3D
MOVL C00099 BC00099 V=500.0  +MOVJ EC00099 VJ=100.00
SMOVL C00100 BC00100 V=100.0  +MOVJ EC00100
SREFP 3 C00101 BC00101  +REFP EC00101
CALL JOB:SEARCH-R1-S13D
SET P033 P006
SFTON3D P033
SMOVL C00102 BC00102 V=100.0  +MOVJ EC00102
SREFP 3 C00103 BC00103  +REFP EC00103
CALL JOB:SEARCH-R1-S13D
SET P033 P006
SFTON3D P033
SMOVL C00104 BC00104 V=100.0  +MOVJ EC00104
MOVL C00105 BC00105 V=833.3  +MOVJ EC00105 VJ=100.00
SMOVL C00106 BC00106 V=100.0  +MOVJ EC00106
SREFP 3 C00107 BC00107  +REFP EC00107
CALL JOB:SEARCH-R1-S13D
SET P034 P006
SFTON3D P034
SMOVL C00108 BC00108 V=100.0  +MOVJ EC00108
SREFP 3 C00109 BC00109  +REFP EC00109
CALL JOB:SEARCH-R1-S13D
SET P034 P006
SFTON3D P034
SMOVL C00110 BC00110 V=100.0  +MOVJ EC00110
MOVL C00111 BC00111 V=1000.0  +MOVJ EC00111 VJ=100.00
MOVJ C00112 BC00112 VJ=100.00  +MOVJ EC00112 VJ=50.00
'Path S1078
SFTOF3D
SMOVL C00113 BC00113 V=133.3  +MOVJ EC00113
SREFP 3 C00114 BC00114  +REFP EC00114
CALL JOB:SEARCH-R1-S13D
SET P035 P006
SFTON3D P035
SMOVL C00115 BC00115 V=100.0  +MOVJ EC00115
SREFP 3 C00116 BC00116  +REFP EC00116
CALL JOB:SEARCH-R1-S13D
SET P035 P006
SFTON3D P035
SMOVL C00117 BC00117 V=100.0  +MOVJ EC00117
MOVL C00118 BC00118 V=400.0  +MOVJ EC00118 VJ=100.00
'Path S1079
SFTOF3D
SMOVL C00119 BC00119 V=166.7  +MOVJ EC00119
SREFP 3 C00120 BC00120  +REFP EC00120
CALL JOB:SEARCH-R1-S13D
SET P036 P006
SFTON3D P036
SMOVL C00121 BC00121 V=100.0  +MOVJ EC00121
SREFP 3 C00122 BC00122  +REFP EC00122
CALL JOB:SEARCH-R1-S13D
SET P036 P006
SFTON3D P036
SMOVL C00123 BC00123 V=100.0  +MOVJ EC00123
MOVJ C00124 BC00124 VJ=100.00  +MOVJ EC00124 VJ=50.00
MOVJ C00125 BC00125 VJ=100.00  +MOVJ EC00125 VJ=50.00
MOVJ C00126 BC00126 VJ=100.00  +MOVJ EC00126 VJ=50.00
MOVJ C00127 BC00127 VJ=100.00  +MOVJ EC00127 VJ=50.00
MOVJ C00128 BC00128 VJ=100.00  +MOVJ EC00128 VJ=50.00
MOVJ C00129 BC00129 VJ=100.00  +MOVJ EC00129 VJ=50.00
SMOVL C00130 BC00130 V=100.0  +MOVJ EC00130
SREFP 3 C00131 BC00131  +REFP EC00131
CALL JOB:SEARCH-R1-S13D
SET P037 P006
SFTON3D P037
SMOVL C00132 BC00132 V=100.0  +MOVJ EC00132
SREFP 3 C00133 BC00133  +REFP EC00133
CALL JOB:SEARCH-R1-S13D
SET P037 P006
SFTON3D P037
SMOVL C00134 BC00134 V=100.0  +MOVJ EC00134
MOVL C00135 BC00135 V=333.3  +MOVJ EC00135 VJ=100.00
'Path S1078
SFTOF3D
SMOVL C00136 BC00136 V=100.0  +MOVJ EC00136
SREFP 3 C00137 BC00137  +REFP EC00137
CALL JOB:SEARCH-R1-S13D
SET P038 P006
SFTON3D P038
SMOVL C00138 BC00138 V=100.0  +MOVJ EC00138
SREFP 3 C00139 BC00139  +REFP EC00139
CALL JOB:SEARCH-R1-S13D
SET P038 P006
SFTON3D P038
SMOVL C00140 BC00140 V=100.0  +MOVJ EC00140
MOVL C00141 BC00141 V=333.3  +MOVJ EC00141 VJ=100.00
'Path S1079
SFTOF3D
MOVL C00142 BC00142 V=400.0  +MOVJ EC00142 VJ=100.00
MOVJ C00143 BC00143 VJ=100.00  +MOVJ EC00143 VJ=50.00
SMOVL C00144 BC00144 V=133.3  +MOVJ EC00144
SREFP 3 C00145 BC00145  +REFP EC00145
CALL JOB:SEARCH-R1-S13D
SET P039 P006
SFTON3D P039
SMOVL C00146 BC00146 V=100.0  +MOVJ EC00146
SREFP 3 C00147 BC00147  +REFP EC00147
CALL JOB:SEARCH-R1-S13D
SET P039 P006
SFTON3D P039
SMOVL C00148 BC00148 V=166.7  +MOVJ EC00148
SFTON3D P039
SMOVL C00149 BC00149 V=166.7 PL=0  +MOVJ EC00149
SREFP 1 C00150 BC00150  +REFP EC00150
SREFP 2 C00151 BC00151  +REFP EC00151
MACRO1 MJ#(0) ARGF14
ARCON
SMOVL C00152 BC00152 V=10.0  +MOVJ EC00152
ARCOF
SFTOF3D
SMOVL C00153 BC00153 V=166.7  +MOVJ EC00153
SMOVL C00154 BC00154 V=416.7  +MOVJ EC00154
SFTOF3D
SFTON3D P037
SMOVL C00155 BC00155 V=133.3 PL=0  +MOVJ EC00155
SREFP 1 C00156 BC00156  +REFP EC00156
SREFP 2 C00157 BC00157  +REFP EC00157
MACRO1 MJ#(0) ARGF17
ARCON
SFTON3D P038
SMOVL C00158 BC00158 V=11.2  +MOVJ EC00158
ARCOF
SFTOF3D
SMOVL C00159 BC00159 V=400.0  +MOVJ EC00159
SMOVL C00160 BC00160 V=250.0  +MOVJ EC00160
MOVJ C00161 BC00161 VJ=100.00  +MOVJ EC00161 VJ=100.00
MOVJ C00162 BC00162 VJ=100.00  +MOVJ EC00162 VJ=100.00
MOVJ C00163 BC00163 VJ=100.00  +MOVJ EC00163 VJ=100.00
MOVJ C00164 BC00164 VJ=100.00  +MOVJ EC00164 VJ=100.00
MOVJ C00165 BC00165 VJ=100.00  +MOVJ EC00165 VJ=100.00
SMOVL C00166 BC00166 V=1000.0  +MOVJ EC00166
SFTOF3D
SFTON3D P032
SMOVL C00167 BC00167 V=133.3 PL=0  +MOVJ EC00167
SREFP 1 C00168 BC00168  +REFP EC00168
SREFP 2 C00169 BC00169  +REFP EC00169
MACRO1 MJ#(0) ARGF14
ARCON
SMOVL C00170 BC00170 V=10.0  +MOVJ EC00170
ARCOF
SMOVL C00171 BC00171 V=400.0  +MOVJ EC00171
SMOVL C00172 BC00172 V=333.3  +MOVJ EC00172
SFTON3D P031
SMOVL C00173 BC00173 V=133.3 PL=0  +MOVJ EC00173
SREFP 1 C00174 BC00174  +REFP EC00174
SREFP 2 C00175 BC00175  +REFP EC00175
MACRO1 MJ#(0) ARGF14
ARCON
SMOVL C00176 BC00176 V=10.0  +MOVJ EC00176
ARCOF
SMOVL C00177 BC00177 V=400.0  +MOVJ EC00177
SMOVL C00178 BC00178 V=250.0  +MOVJ EC00178
SFTON3D P034
SMOVL C00179 BC00179 V=133.3 PL=0  +MOVJ EC00179
SREFP 1 C00180 BC00180  +REFP EC00180
SREFP 2 C00181 BC00181  +REFP EC00181
MACRO1 MJ#(0) ARGF14
ARCON
SMOVL C00182 BC00182 V=10.0  +MOVJ EC00182
ARCOF
SMOVL C00183 BC00183 V=400.0  +MOVJ EC00183
SMOVL C00184 BC00184 V=666.7  +MOVJ EC00184
SFTON3D P033
SMOVL C00185 BC00185 V=133.3 PL=0  +MOVJ EC00185
SREFP 1 C00186 BC00186  +REFP EC00186
SREFP 2 C00187 BC00187  +REFP EC00187
MACRO1 MJ#(0) ARGF14
ARCON
SMOVL C00188 BC00188 V=10.0  +MOVJ EC00188
ARCOF
SMOVL C00189 BC00189 V=1000.0  +MOVJ EC00189
SMOVL C00190 BC00190 V=500.0  +MOVJ EC00190
SFTON3D P036
SMOVL C00191 BC00191 V=133.3 PL=0  +MOVJ EC00191
SREFP 1 C00192 BC00192  +REFP EC00192
SREFP 2 C00193 BC00193  +REFP EC00193
MACRO1 MJ#(0) ARGF14
ARCON
SMOVL C00194 BC00194 V=10.0  +MOVJ EC00194
ARCOF
SMOVL C00195 BC00195 V=400.0  +MOVJ EC00195
SMOVL C00196 BC00196 V=500.0  +MOVJ EC00196
'SPRAWDZIC SPOINE
SFTON3D P035
SMOVL C00197 BC00197 V=133.3 PL=0  +MOVJ EC00197
SREFP 1 C00198 BC00198  +REFP EC00198
SREFP 2 C00199 BC00199  +REFP EC00199
MACRO1 MJ#(0) ARGF14
ARCON
SMOVL C00200 BC00200 V=10.0  +MOVJ EC00200
ARCOF
SMOVL C00201 BC00201 V=666.7  +MOVJ EC00201
MOVJ C00202 BC00202 VJ=100.00  +MOVJ EC00202 VJ=50.00
'obrot
MOVJ C00203 BC00203 VJ=100.00  +MOVJ EC00203 VJ=100.00
MOVJ C00204 BC00204 VJ=100.00  +MOVJ EC00204 VJ=100.00
MOVJ C00205 BC00205 VJ=100.00  +MOVJ EC00205 VJ=100.00
MOVJ C00206 BC00206 VJ=100.00  +MOVJ EC00206 VJ=100.00
MOVJ C00207 BC00207 VJ=100.00  +MOVJ EC00207 VJ=100.00
MOVJ C00208 BC00208 VJ=100.00  +MOVJ EC00208 VJ=100.00
MOVJ C00209 BC00209 VJ=100.00  +MOVJ EC00209 VJ=100.00
'Path W1425
SFTOF3D
SFTON3D P023
MOVJ C00210 BC00210 VJ=100.00  +MOVJ EC00210 VJ=100.00
SMOVL C00211 BC00211 V=333.3  +MOVJ EC00211
SMOVL C00212 BC00212 V=133.3 PL=0  +MOVJ EC00212
SREFP 1 C00213 BC00213  +REFP EC00213
SREFP 2 C00214 BC00214  +REFP EC00214
MACRO1 MJ#(0) ARGF14
ARCON
SMOVL C00215 BC00215 V=10.0  +MOVJ EC00215
ARCOF
SMOVL C00216 BC00216 V=400.0  +MOVJ EC00216
SMOVL C00217 BC00217 V=1000.0  +MOVJ EC00217
SFTOF3D
SFTON3D P022
MOVJ C00218 BC00218 VJ=100.00  +MOVJ EC00218 VJ=100.00
SMOVL C00219 BC00219 V=133.3 PL=0  +MOVJ EC00219
SREFP 1 C00220 BC00220  +REFP EC00220
SREFP 2 C00221 BC00221  +REFP EC00221
MACRO1 MJ#(0) ARGF14
ARCON
SMOVL C00222 BC00222 V=10.0  +MOVJ EC00222
ARCOF
SMOVL C00223 BC00223 V=400.0  +MOVJ EC00223
SMOVL C00224 BC00224 V=1000.0  +MOVJ EC00224
SFTOF3D
SFTON3D P021
MOVJ C00225 BC00225 VJ=100.00  +MOVJ EC00225 VJ=100.00
SMOVL C00226 BC00226 V=133.3 PL=0  +MOVJ EC00226
SREFP 1 C00227 BC00227  +REFP EC00227
SREFP 2 C00228 BC00228  +REFP EC00228
MACRO1 MJ#(0) ARGF14
ARCON
SMOVL C00229 BC00229 V=10.0  +MOVJ EC00229
ARCOF
SMOVL C00230 BC00230 V=400.0  +MOVJ EC00230
SMOVL C00231 BC00231 V=333.3  +MOVJ EC00231
SFTON3D P026
SMOVL C00232 BC00232 V=133.3 PL=0  +MOVJ EC00232
SREFP 1 C00233 BC00233  +REFP EC00233
SREFP 2 C00234 BC00234  +REFP EC00234
MACRO1 MJ#(0) ARGF14
ARCON
SMOVL C00235 BC00235 V=10.0  +MOVJ EC00235
ARCOF
SMOVL C00236 BC00236 V=400.0  +MOVJ EC00236
SMOVL C00237 BC00237 V=1000.0  +MOVJ EC00237
SFTOF3D
SFTON3D P025
SMOVL C00238 BC00238 V=133.3 PL=0  +MOVJ EC00238
SREFP 1 C00239 BC00239  +REFP EC00239
SREFP 2 C00240 BC00240  +REFP EC00240
MACRO1 MJ#(0) ARGF14
ARCON
SMOVL C00241 BC00241 V=10.0  +MOVJ EC00241
ARCOF
SMOVL C00242 BC00242 V=400.0  +MOVJ EC00242
SMOVL C00243 BC00243 V=1000.0  +MOVJ EC00243
SFTOF3D
'Path W1427
SFTOF3D
SFTON3D P024
SMOVL C00244 BC00244 V=133.3 PL=0  +MOVJ EC00244
SREFP 1 C00245 BC00245  +REFP EC00245
SREFP 2 C00246 BC00246  +REFP EC00246
MACRO1 MJ#(0) ARGF14
ARCON
SMOVL C00247 BC00247 V=10.0  +MOVJ EC00247
ARCOF
SMOVL C00248 BC00248 V=400.0  +MOVJ EC00248
MOVJ C00249 BC00249 VJ=100.00  +MOVJ EC00249 VJ=100.00
MOVJ C00250 BC00250 VJ=100.00  +MOVJ EC00250 VJ=100.00
MOVJ C00251 BC00251 VJ=100.00  +MOVJ EC00251 VJ=100.00
MOVJ C00252 BC00252 VJ=100.00  +MOVJ EC00252 VJ=100.00
MOVJ C00253 BC00253 VJ=100.00  +MOVJ EC00253 VJ=100.00
MOVJ C00254 BC00254 VJ=100.00  +MOVJ EC00254 VJ=100.00
SFTON3D P027
SMOVL C00255 BC00255 V=166.7  +MOVJ EC00255
ARCON
SMOVL C00256 BC00256 V=10.0  +MOVJ EC00256
ARCOF
SFTOF3D
MOVJ C00257 BC00257 VJ=100.00  +MOVJ EC00257 VJ=100.00
MOVJ C00258 BC00258 VJ=100.00  +MOVJ EC00258 VJ=100.00
MOVJ C00259 BC00259 VJ=100.00  +MOVJ EC00259 VJ=100.00
SFTON3D P030
SMOVL C00260 BC00260 V=133.3  +MOVJ EC00260
ARCON
SFTON3D P029
SMOVL C00261 BC00261 V=10.0  +MOVJ EC00261
ARCOF
SFTOF3D
SMOVL C00262 BC00262 V=250.0  +MOVJ EC00262
MOVJ C00263 BC00263 VJ=100.00  +MOVJ EC00263 VJ=100.00
MOVJ C00264 BC00264 VJ=100.00  +MOVJ EC00264 VJ=100.00
MOVJ C00265 BC00265 VJ=100.00  +MOVJ EC00265 VJ=100.00
'KONIEC
END
